// TIA Portal V17 export
// export: Created 2023-02-14T02:49:31.443303Z, ExportSetting WithDefaults, DisplayName Totally Integrated Automation Portal, DisplayVersion V17, DisplayName TIA Portal Openness, DisplayVersion V17, DisplayName TIA Portal Teamcenter Gateway, DisplayVersion V17, DisplayName TIA Portal Version Control Interface, DisplayVersion V17, DisplayName SINAMICS Startdrive Advanced, DisplayVersion V17, DisplayName SINAMICS Startdrive G130, G150, S120, S150, SINAMICS MV, S210, DisplayVersion V17, DisplayName SINAMICS Startdrive G110M, G120, G120C, G120D, G120P, G115D, DisplayVersion V17, DisplayName STEP 7 Professional, DisplayVersion V17, DisplayName STEP 7 Safety, DisplayVersion V17, DisplayName WinCC Professional, DisplayVersion V17
DATA_BLOCK "IO_Digital_Storage_DB"   // DB44
VERSION : 0.1
// stored: AutoNumber true, DBAccessibleFromOPCUA true, DBAccessibleFromWebserver true, InstanceOfName IO_Digital_Storage, InstanceOfType FB
"IO_Digital_Storage"
   // VAR_INPUT
   //    lock : Bool;
   //    init : Bool;
   //    Reset : Bool;
   // END_VAR
   // VAR
   //    "FS-23.01" : "Digital";
   //    "FS-24.01" { S7_SetPoint := 'True'} : "Digital";
   //    "FS-34.01" { S7_SetPoint := 'True'} : "Digital";
   //    "FS-35.01" { S7_SetPoint := 'True'} : "Digital";
   // END_VAR
BEGIN
END_DATA_BLOCK
